Staubli VAL3: exeSearchL.pgx

program exeSearchL(dio x_dInput, tool x_tTool)
begin

  wait(x_dInput==true or bSearchLFail)
  if x_dInput==true
    resetMotion()
    bSearchLSuccess=true
  else
    logMsg("libSignals/exeSearchL->timeout")
  endIf

end
